(* Logix 5000 project; controller VFX vendor 1 type 14 code 177 rev 31.11; software revision 31.00; part 2 of 2 *)
(* tags used below, declared in another part *)
   boxtypes : BOXTYPE[10];
   fanuc : FANUC_MASTER;
   fanuc_IPC_start : BOOL;
   fanuc_s1 : FANUC_EDA_T;
   fanuc_style_start : BOOL;
   fanuc_target_boxtype : DINT;
   out_fail2 : BOOL;
   out_pass2 : BOOL;
   output_pulse2 : DINT;
   step_robot_command : DINT;
   tmr_pulse_fanuc : TIMER;
   tmr_pulse_fanuc_done : TIMER;
   tmr_start_fanuc : TIMER;
(* VFX, continued *)

ROUTINE fanuc_logic   (* ladder *)
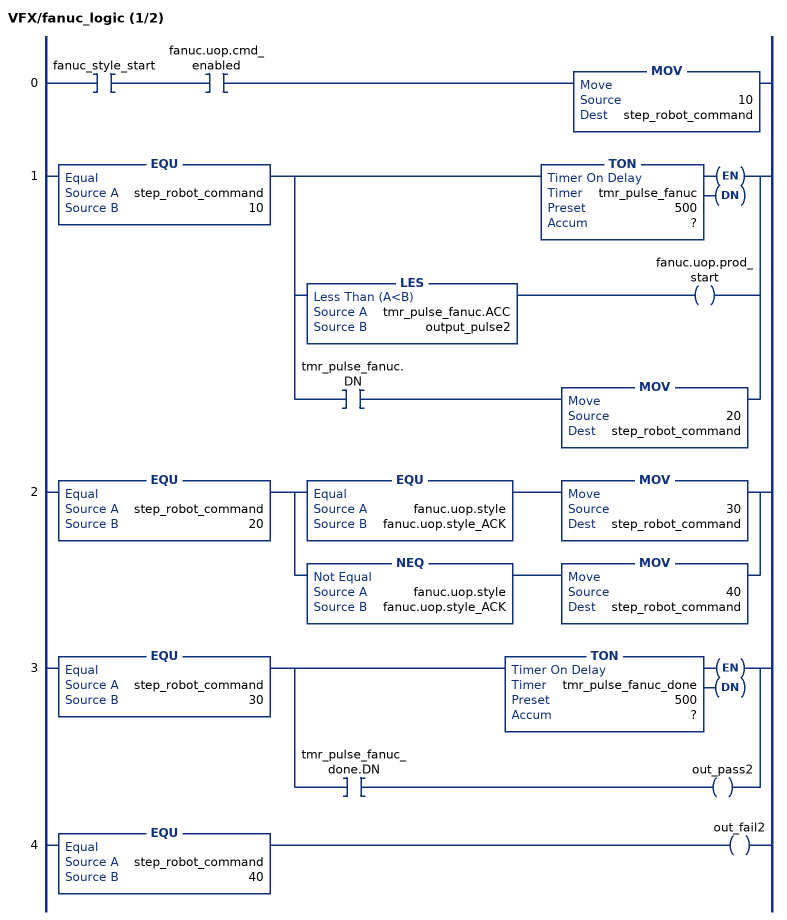
   0: XIC(fanuc_style_start)XIC(fanuc.uop.cmd_enabled)MOV(10,step_robot_command);
   1: EQU(step_robot_command,10)[TON(tmr_pulse_fanuc,?,?) ,LES(tmr_pulse_fanuc.ACC,output_pulse2) OTE(fanuc.uop.prod_start) ,XIC(tmr_pulse_fanuc.DN) MOV(20,step_robot_command) ];
   2: EQU(step_robot_command,20)[EQU(fanuc.uop.style,fanuc.uop.style_ACK) MOV(30,step_robot_command) ,NEQ(fanuc.uop.style,fanuc.uop.style_ACK) MOV(40,step_robot_command) ];
   3: EQU(step_robot_command,30)[TON(tmr_pulse_fanuc_done,?,?) ,XIC(tmr_pulse_fanuc_done.DN) OTE(out_pass2) ];
   4: EQU(step_robot_command,40)OTE(out_fail2);
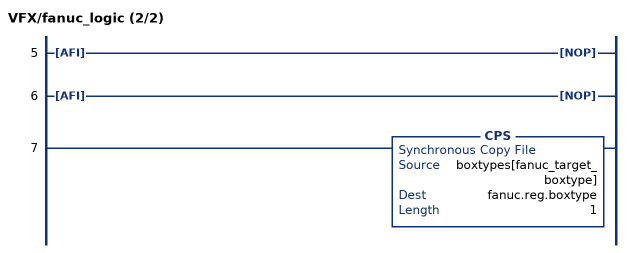
   5: AFI()NOP();
   6: AFI()NOP();
   7: CPS(boxtypes[fanuc_target_boxtype],fanuc.reg.boxtype,1);
END_ROUTINE

ROUTINE IPC_IO   (* ladder *)
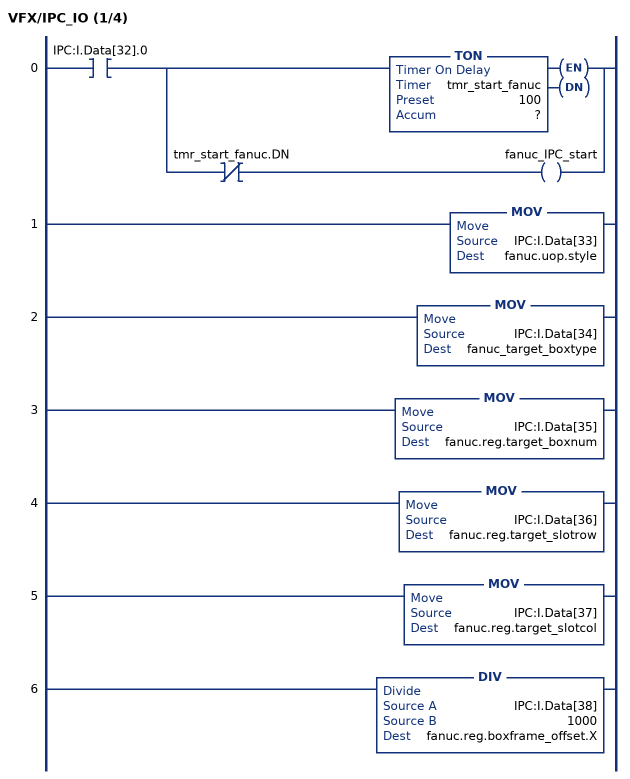
   0: XIC(IPC:I.Data[32].0)[TON(tmr_start_fanuc,?,?) ,XIO(tmr_start_fanuc.DN) OTE(fanuc_IPC_start) ];
   1: MOV(IPC:I.Data[33],fanuc.uop.style);
   2: MOV(IPC:I.Data[34],fanuc_target_boxtype);
   3: MOV(IPC:I.Data[35],fanuc.reg.target_boxnum);
   4: MOV(IPC:I.Data[36],fanuc.reg.target_slotrow);
   5: MOV(IPC:I.Data[37],fanuc.reg.target_slotcol);
   6: DIV(IPC:I.Data[38],1000,fanuc.reg.boxframe_offset.X);
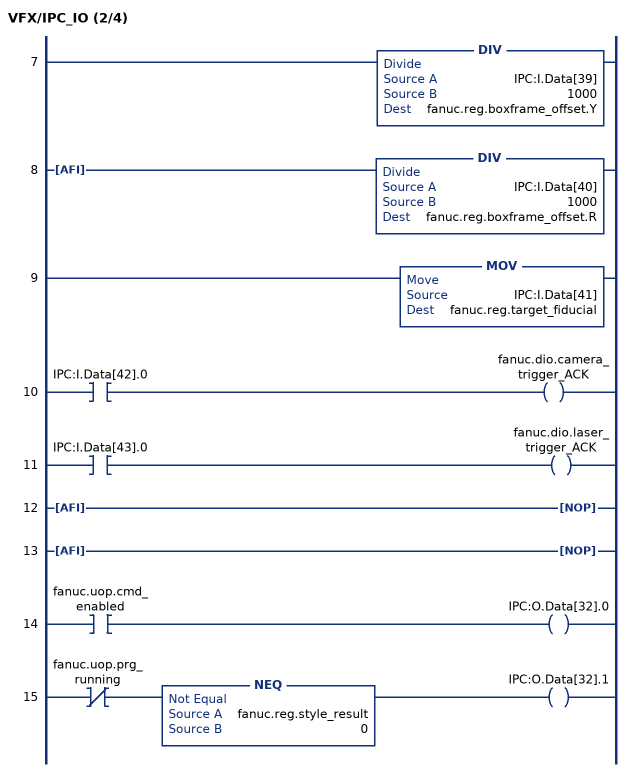
   7: DIV(IPC:I.Data[39],1000,fanuc.reg.boxframe_offset.Y);
   8: AFI()DIV(IPC:I.Data[40],1000,fanuc.reg.boxframe_offset.R);
   9: MOV(IPC:I.Data[41],fanuc.reg.target_fiducial);
   10: XIC(IPC:I.Data[42].0)OTE(fanuc.dio.camera_trigger_ACK);
   11: XIC(IPC:I.Data[43].0)OTE(fanuc.dio.laser_trigger_ACK);
   12: AFI()NOP();
   13: AFI()NOP();
   14: XIC(fanuc.uop.cmd_enabled)OTE(IPC:O.Data[32].0);
   15: XIO(fanuc.uop.prg_running)NEQ(fanuc.reg.style_result,0)OTE(IPC:O.Data[32].1);
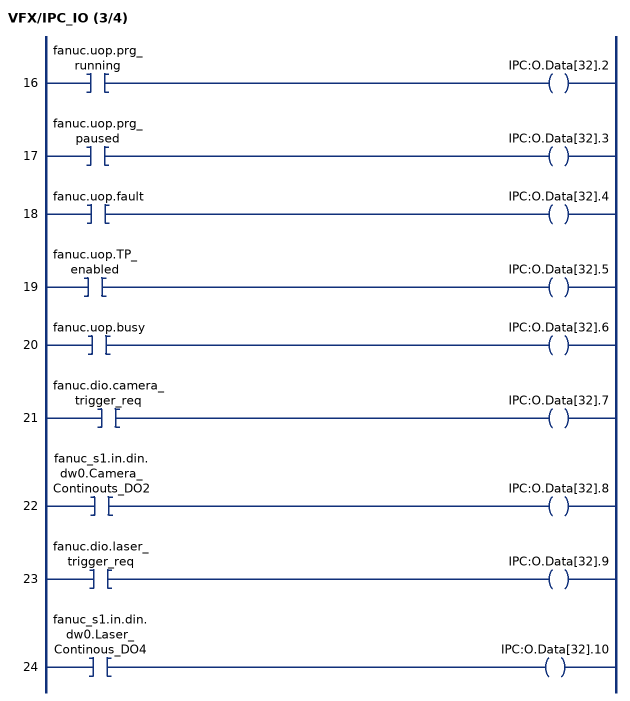
   16: XIC(fanuc.uop.prg_running)OTE(IPC:O.Data[32].2);
   17: XIC(fanuc.uop.prg_paused)OTE(IPC:O.Data[32].3);
   18: XIC(fanuc.uop.fault)OTE(IPC:O.Data[32].4);
   19: XIC(fanuc.uop.TP_enabled)OTE(IPC:O.Data[32].5);
   20: XIC(fanuc.uop.busy)OTE(IPC:O.Data[32].6);
   21: XIC(fanuc.dio.camera_trigger_req)OTE(IPC:O.Data[32].7);
   22: XIC(fanuc_s1.in.din.dw0.Camera_Continouts_DO2)OTE(IPC:O.Data[32].8);
   23: XIC(fanuc.dio.laser_trigger_req)OTE(IPC:O.Data[32].9);
   24: XIC(fanuc_s1.in.din.dw0.Laser_Continous_DO4)OTE(IPC:O.Data[32].10);
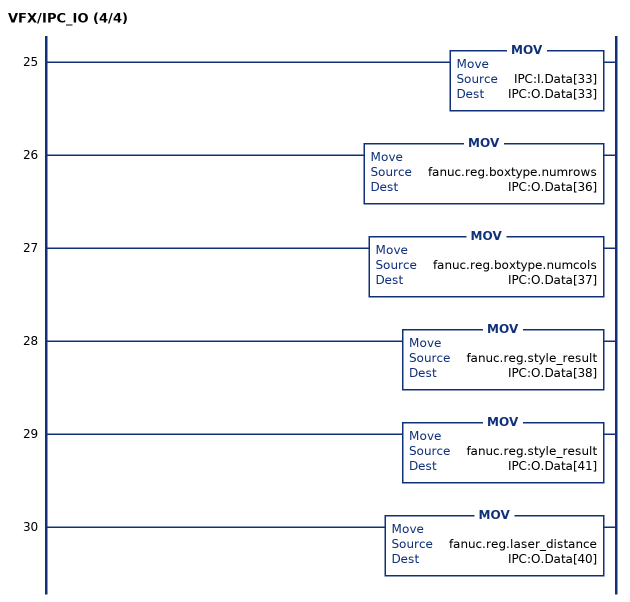
   25: MOV(IPC:I.Data[33],IPC:O.Data[33]);
   26: MOV(fanuc.reg.boxtype.numrows,IPC:O.Data[36]);
   27: MOV(fanuc.reg.boxtype.numcols,IPC:O.Data[37]);
   28: MOV(fanuc.reg.style_result,IPC:O.Data[38]);
   29: MOV(fanuc.reg.style_result,IPC:O.Data[41]);
   30: MOV(fanuc.reg.laser_distance,IPC:O.Data[40]);
END_ROUTINE

ROUTINE MainRoutine   (* ladder *)
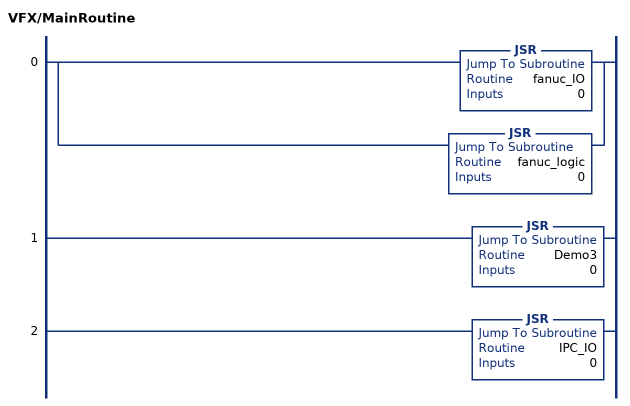
   0: [JSR(fanuc_IO,0) ,JSR(fanuc_logic,0) ];
   1: JSR(Demo3,0);
   2: JSR(IPC_IO,0);
END_ROUTINE
END_PROGRAM
